# B&R Automation Studio project git_1
Automation Studio 4.6.3.55

## Configuration Config1

### Task classes (Cpu.sw)
```

```

### Hardware
```
X20CP1586 : X20CP1586 v1.5.0.0
```

## Logical view

### RevInfo.var
```iecst
VAR CONSTANT
	revision : STRING[80] := '';
	revisionDate : STRING[80] := '';
	revisionAuthor : STRING[80] := '';
	branchName : STRING[80] := '';
	uncommittedChanges : STRING[80] := '';
	buildDate  : STRING[80] := '2022-04-22 11:26:09 +0800';
	buildConfiguration : STRING[80] := '';
	builder : STRING[80] := '';
END_VAR
```
